// TIA Portal V17 export
// export: Created 2026-04-13T11:12:53.4843074Z, ExportSetting WithDefaults, DisplayName Totally Integrated Automation Portal, DisplayVersion V17 Update 4, DisplayName TIA Portal Openness, DisplayVersion V17 Update 4, DisplayName TIA Portal Version Control Interface, DisplayVersion V17, DisplayName SINAMICS Startdrive Advanced, DisplayVersion V17, DisplayName SINAMICS Startdrive G130, G150, S120, S150, SINAMICS MV, S210, DisplayVersion V17, DisplayName SINAMICS Startdrive G110M, G120, G120C, G120D, G120P, G115D, DisplayVersion V17, DisplayName STEP 7 Professional, DisplayVersion V17 Update 4, DisplayName STEP 7 Safety, DisplayVersion V17, DisplayName WinCC Professional, DisplayVersion V17 Update 4
TagTable "INCIPRJ"
  INCIPRJ_1设定时间 : Real  (PLC tag INCIPRJ.1设定时间, HMI_连接_1, 1 s)
  INCIPRJ_2设定时间 : Real  (PLC tag INCIPRJ.2设定时间, HMI_连接_1, 1 s)
  INCIPRJ_3设定时间 : Real  (PLC tag INCIPRJ.3设定时间, HMI_连接_1, 1 s)
  INCIPRJ_4设定时间 : Real  (PLC tag INCIPRJ.4设定时间, HMI_连接_1, 1 s)
  INCIPRJ_5设定时间 : Real  (PLC tag INCIPRJ.5设定时间, HMI_连接_1, 1 s)
  INCIPRJ_6设定时间 : Real  (PLC tag INCIPRJ.6设定时间, HMI_连接_1, 1 s)
  INCIPRJ_7设定时间 : Real  (PLC tag INCIPRJ.7设定时间, HMI_连接_1, 1 s)
  INCIPRJ_8设定时间 : Real  (PLC tag INCIPRJ.8设定时间, HMI_连接_1, 1 s)
  INCIPRJ_9设定时间 : Real  (PLC tag INCIPRJ.9设定时间, HMI_连接_1, 1 s)
  INCIPRJ_10设定时间 : Real  (PLC tag INCIPRJ.10设定时间, HMI_连接_1, 1 s)
  INCIPRJ_11设定时间 : Real  (PLC tag INCIPRJ.11设定时间, HMI_连接_1, 1 s)
  INCIPRJ_12设定时间 : Real  (PLC tag INCIPRJ.12设定时间, HMI_连接_1, 1 s)
  INCIPRJ_13设定时间 : Real  (PLC tag INCIPRJ.13设定时间, HMI_连接_1, 1 s)
  INCIPRJ_14设定时间 : Real  (PLC tag INCIPRJ.14设定时间, HMI_连接_1, 1 s)
  INCIPRJ_15设定时间 : Real  (PLC tag INCIPRJ.15设定时间, HMI_连接_1, 1 s)
  INCIPRJ_16设定时间 : Real  (PLC tag INCIPRJ.16设定时间, HMI_连接_1, 1 s)
  INCIPRJ_1计时 : Real  (PLC tag INCIPRJ.1计时, HMI_连接_1, 1 s)
  INCIPRJ_2计时 : Real  (PLC tag INCIPRJ.2计时, HMI_连接_1, 1 s)
  INCIPRJ_3计时 : Real  (PLC tag INCIPRJ.3计时, HMI_连接_1, 1 s)
  INCIPRJ_4计时 : Real  (PLC tag INCIPRJ.4计时, HMI_连接_1, 1 s)
  INCIPRJ_5计时 : Real  (PLC tag INCIPRJ.5计时, HMI_连接_1, 1 s)
  INCIPRJ_6计时 : Real  (PLC tag INCIPRJ.6计时, HMI_连接_1, 1 s)
  INCIPRJ_7计时 : Real  (PLC tag INCIPRJ.7计时, HMI_连接_1, 1 s)
  INCIPRJ_8计时 : Real  (PLC tag INCIPRJ.8计时, HMI_连接_1, 1 s)
  INCIPRJ_9计时 : Real  (PLC tag INCIPRJ.9计时, HMI_连接_1, 1 s)
  INCIPRJ_10计时 : Real  (PLC tag INCIPRJ.10计时, HMI_连接_1, 1 s)
  INCIPRJ_11计时 : Real  (PLC tag INCIPRJ.11计时, HMI_连接_1, 1 s)
  INCIPRJ_12计时 : Real  (PLC tag INCIPRJ.12计时, HMI_连接_1, 1 s)
  INCIPRJ_13计时 : Real  (PLC tag INCIPRJ.13计时, HMI_连接_1, 1 s)
  INCIPRJ_14计时 : Real  (PLC tag INCIPRJ.14计时, HMI_连接_1, 1 s)
  INCIPRJ_15计时 : Real  (PLC tag INCIPRJ.15计时, HMI_连接_1, 1 s)
  INCIPRJ_16计时 : Real  (PLC tag INCIPRJ.16计时, HMI_连接_1, 1 s)
